FUNCTION_BLOCK FB_PerMCS2MotorFFOND
(*
    PMPS fast faults that must be done per motor, rather than per state, based purely
    on the motor status and not other PMPS considerations.

    These currently include:
    - Fault if the encoder has an error. Every other protection is based on the encoder,
      so we can't trust anything if the encoder is faulting.
*)
VAR_IN_OUT
    // All motors associated with the state mover.
    astMotionStage: ARRAY[1..MotionConstants.MAX_STATE_MOTORS] OF ST_MCS2Stage;
    // Fast fault output to fault to.
    fbFFHWO: FB_HardwareFFOutput;
END_VAR
VAR_INPUT
    // The number of motors we're actually using
    nActiveMotorCount: UINT;
    // Identifying name to use in group fast faults
    sDeviceName: STRING;
END_VAR
VAR_OUTPUT
    // Set to TRUE if the arrays don't have the same bounds. In this FB, that's an automatic fault.
    bMotorCountError: BOOL;
END_VAR
VAR
    afbEncError: ARRAY[1..MotionConstants.MAX_STATE_MOTORS] OF FB_EncErrorFFO;
    ffProgrammerError: FB_FastFault;
    nIter: DINT;
END_VAR

// Make sure the motor count is valid (positive, nonzero, less or equal to the max)
bMotorCountError S= nActiveMotorCount <= 0;
bMotorCountError S= nActiveMotorCount > MotionConstants.MAX_STATE_MOTORS;

IF NOT bMotorCountError THEN
    // Handle Loop
    FOR nIter := 1 TO nActiveMotorCount DO
        afbEncError[nIter](
            stMotionstage:=astMotionStage[nIter],
            fbFFHWO:=fbFFHWO,
            bAutoReset:=TRUE,
        );
    END_FOR
END_IF
// handle FFO
ffProgrammerError(
    i_xOK:=NOT bMotorCountError,
    i_xAutoReset:=TRUE,
    i_DevName:=sDeviceName,
    i_Desc:='Programmer error picking motor count',
    i_TypeCode:=E_MotionFFType.INTERNAL_ERROR,
    io_fbFFHWO:=fbFFHWO,
);

END_FUNCTION_BLOCK

(* stored: Version 1.1.0.1
   POU FB_PerMCS2MotorFFOND: Id {244016c5-5c36-491e-aa05-49dc353243ed}, SpecialFunc None *)
